# EPICS substitutions: apps/caen1527App/Db/user.substitutions
# Example substitutions file

file "db/circle.db" {
    { user = "bbhodo" }
}

file "db/dbExample1.db" {
    { user = "bbhodo" }
}

file db/dbExample2.db {
    pattern { user, no, scan }
        { "bbhodo", 1, "1 second" }
        { "bbhodo", 2, "2 second" }
        { "bbhodo", 3, "5 second" }
}
